// TIA Portal V16 export
// export: Created 2021-12-01T21:19:41.5280979Z, ExportSetting WithDefaults, DisplayName Totally Integrated Automation Portal, DisplayVersion V16 Update 4, DisplayName TIA Portal Version Control Interface, DisplayVersion V16 Update 2, DisplayName TIA Portal Openness, DisplayVersion V16 Update 4, DisplayName SINAMICS Startdrive Advanced, DisplayVersion V16 Update 5, DisplayName SINAMICS Startdrive G130, G150, S120, S150, SINAMICS MV, S210, DisplayVersion V16 Update 5, DisplayName SINAMICS Startdrive G110M, G120, G120C, G120D, G120P, G115D, DisplayVersion V16 Update 5, DisplayName STEP 7 Professional, DisplayVersion V16 Update 4, DisplayName STEP 7 Safety, DisplayVersion V16, DisplayName WinCC Advanced, DisplayVersion V16 Update 4
DATA_BLOCK "ST00315_PLTCP_SL_UDT2100_IDB"   // DB529
VERSION : 0.1
// stored: AutoNumber true, DBAccessibleFromOPCUA true, InstanceOfName PLTCPsendReceive_1, InstanceOfType FB
"PLTCPsendReceive_1"
   // VAR_INPUT
   //    Enable { ExternalAccessible := 'False'; ExternalVisible := 'False'; ExternalWritable := 'False'} : Bool;
   //    UDTnumber { ExternalAccessible := 'False'; ExternalVisible := 'False'; ExternalWritable := 'False'} : UInt;
   //    UDTversion { ExternalAccessible := 'False'; ExternalVisible := 'False'; ExternalWritable := 'False'} : UInt;
   //    ExpectedUDTnumber { ExternalAccessible := 'False'; ExternalVisible := 'False'; ExternalWritable := 'False'} : UInt;
   //    ExpectedUDTversion { ExternalAccessible := 'False'; ExternalVisible := 'False'; ExternalWritable := 'False'} : UInt;
   //    UniqeID { ExternalAccessible := 'False'; ExternalVisible := 'False'; ExternalWritable := 'False'} : String["Const_PLTCP_UniqueIDSize"];
   //    Trigger { ExternalAccessible := 'False'; ExternalVisible := 'False'; ExternalWritable := 'False'} : Bool;
   //    TriggerOnly { ExternalAccessible := 'False'; ExternalVisible := 'False'; ExternalWritable := 'False'} : Bool;
   //    UDTtoClient : Variant;
   // END_VAR
   // VAR_OUTPUT
   //    SendStatus { ExternalAccessible := 'False'; ExternalVisible := 'False'; ExternalWritable := 'False'} : SInt;
   //    NewMessageReceived { ExternalAccessible := 'False'; ExternalVisible := 'False'; ExternalWritable := 'False'} : Bool;
   //    Error { ExternalAccessible := 'False'; ExternalVisible := 'False'; ExternalWritable := 'False'} : "UDT_Error";
   // END_VAR
   // VAR_IN_OUT
   //    UDTfromClient : Variant;
   // END_VAR
   // VAR
   //    MessageConstructor_Single { ExternalAccessible := 'False'; ExternalVisible := 'False'; ExternalWritable := 'False'} : "MessageConstructor_Single_1";
   //    DestructorWhileLoopTime { ExternalAccessible := 'False'; ExternalVisible := 'False'; ExternalWritable := 'False'} : LTime;
   //    MessageConstructorUDT5_Single { ExternalAccessible := 'False'; ExternalVisible := 'False'; ExternalWritable := 'False'} : "MessageConstructorUDT5_Single_2";
   //    ClientRequest { ExternalAccessible := 'False'; ExternalVisible := 'False'; ExternalWritable := 'False'} : "UDT_ClientRequest";
   //    Ons { ExternalAccessible := 'False'; ExternalVisible := 'False'; ExternalWritable := 'False'} : Array[0..10] of Bool;
   //    SubscribeAcknowledged { ExternalAccessible := 'False'; ExternalVisible := 'False'; ExternalWritable := 'False'} : Bool;
   // END_VAR
BEGIN
END_DATA_BLOCK
